KUKA KRL program: Circular.src, Circular.dat

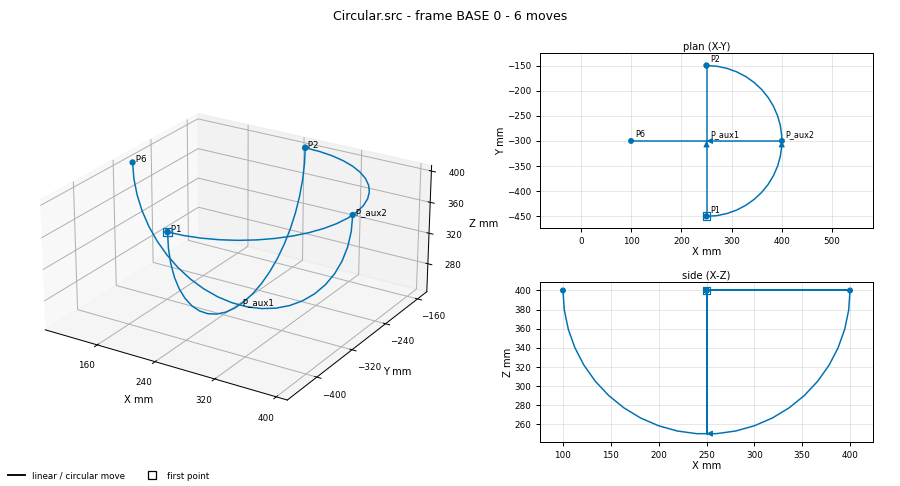
[picture p0: tool path of Circular.src in frame BASE 0, 6 of 10 moves have a stored position in this frame; points joined in program order, loops and branches not executed]
--- Circular.src ---
&ACCESS RVO
&REL 2
&PARAM DISKPATH = KRC:\R1\Program\My_Project
DEF  Circular ( )
;FOLD INI;%{PE}
  ;FOLD BASISTECH INI
    GLOBAL INTERRUPT DECL 3 WHEN $STOPMESS==TRUE DO IR_STOPM ( )
    INTERRUPT ON 3
    BAS (#INITMOV,0 )
  ;ENDFOLD (BASISTECH INI)
  ;FOLD USER INI
    ;Make your modifications here

  ;ENDFOLD (USER INI)
;ENDFOLD (INI)

;FOLD SPTP HOME Vel=100 % DEFAULT ;%{PE}
;FOLD Parameters ;%{h}
;Params IlfProvider=kukaroboter.basistech.inlineforms.movement.spline; Kuka.IsGlobalPoint=False; Kuka.PointName=HOME; Kuka.BlendingEnabled=False; Kuka.MoveDataPtpName=DEFAULT; Kuka.VelocityPtp=100; Kuka.VelocityFieldEnabled=True; Kuka.CurrentCDSetIndex=0; Kuka.MovementParameterFieldEnabled=True; IlfCommand=SPTP
;ENDFOLD
PTP XHOME                                              ;Go to Home position
;ENDFOLD

$BWDSTART = FALSE
PDAT_ACT = PPDATP
FDAT_ACT = FP
BAS(#PTP_PARAMS, 100)
SET_CD_PARAMS(0)


PTP P1                                            ;PTP movement to Point P1
$CIRC_TYPE = #BASE                                ;Set control of circular movement to be BASE related
$ORI_TYPE = #CONSTANT                             ;Set Orientation of the TCP to be CONSTANT
TraceStart("New_KSS_8.5_1.xml", "roll")           ;Start recording trace with the mentioned Trace configuration
CIRC P_aux1, P2, CA 360.0
TraceStop()
PTP XHOME

PTP P3                                            ;PTP movement to Point P3
$CIRC_TYPE = #BASE                                ;Set control of circular movement to be BASE related
$ORI_TYPE = #CONSTANT                             ;Set Orientation of the TCP to be CONSTANT
TraceStart("New_KSS_8.5_1.xml", "yaw")            ;Start recording trace with the mentioned Trace configuration
CIRC P_aux2, P4, CA 360.0
TraceStop()
PTP XHOME

PTP P5                                            ;PTP movement to Point P5
$CIRC_TYPE = #BASE                                ;Set control of circular movement to be BASE related
$ORI_TYPE = #CONSTANT                             ;Set Orientation of the TCP to be CONSTANT
TraceStart("New_KSS_8.5_1.xml", "pitch")          ;Start recording trace with the mentioned Trace configuration
CIRC P_aux3, P6, CA 360.0
TraceStop()

;FOLD SPTP HOME Vel=100 % DEFAULT ;%{PE}
;FOLD Parameters ;%{h}
;Params IlfProvider=kukaroboter.basistech.inlineforms.movement.spline; Kuka.IsGlobalPoint=False; Kuka.PointName=HOME; Kuka.BlendingEnabled=False; Kuka.MoveDataPtpName=DEFAULT; Kuka.VelocityPtp=100; Kuka.VelocityFieldEnabled=True; Kuka.CurrentCDSetIndex=0; Kuka.MovementParameterFieldEnabled=True; IlfCommand=SPTP
;ENDFOLD
PTP XHOME                                              ;Go to Home position
;ENDFOLD

END

--- Circular.dat ---
&ACCESS RVO
&REL 2
&PARAM DISKPATH = KRC:\R1\Program\My_Project
DEFDAT Circular
;FOLD EXTERNAL DECLARATIONS;%{PE}%MKUKATPBASIS,%CEXT,%VCOMMON,%P
;FOLD BASISTECH EXT;%{PE}%MKUKATPBASIS,%CEXT,%VEXT,%P
EXT  BAS (BAS_COMMAND  :IN,REAL  :IN )
DECL INT SUCCESS
;ENDFOLD (BASISTECH EXT)
;FOLD USER EXT;%{E}%MKUKATPUSER,%CEXT,%VEXT,%P
;Make your modifications here

DECL E6AXIS XHOME = {A1 0.0, A2 -110.0, A3 110.0, A4 0.0, A5 0.0, A6 0.0}                  ;Home Position

DECL PDAT PPDATP={VEL 100.000,ACC 100.000,APO_DIST 100.000,APO_MODE #CDIS,GEAR_JERK 100.000,EXAX_IGN 0}     ;Set the kinematic values such as max velocity, max acceleration, etc
DECL FDAT FP={TOOL_NO 14,BASE_NO 0,IPO_FRAME #BASE,POINT2[] " ",TQ_STATE FALSE}                             ;Set the tool and base for coordinate transformation

DECL E6POS P1 = {X 250.0, Y -450.0, Z 400.0, A 0.0, B 45, C 0.0, S 2, T 10}                 ;Point P1
DECL E6POS P_aux1 = {X 250.0, Y -300.0, Z 250.0, A 0.0, B 45, C 0.0, S 2, T 10}             ;Point P_aux1
DECL E6POS P2 = {X 250.0, Y -150.0, Z 400.0, A 0.0, B 45, C 0.0, S 2, T 10}                 ;Point P2

DECL E6POS P3 = {X 250.0, Y -450.0, Z 400.0, A -12.32, B 82.93, C -12.5, S 2, T 10}         ;Point P3
DECL E6POS P_aux2 = {X 400.0, Y -300.0, Z 400.0, A -12.32, B 82.93, C -12.5, S 2, T 10}     ;Point P_aux2
DECL E6POS P4 = {X 250.0, Y -150.0, Z 400.0, A -12.32, B 82.93, C -12.5, S 2, T 10}         ;Point P4

DECL E6POS P5 = {X 400.0, Y -300.0, Z 400.0, A 0.0, B 45.0, C 0.0, S 2, T 10}               ;Point P5
DECL E6POS P_aux3 = {X 250.0, Y -300.0, Z 250.0, A 0.0, B 45.0, C 0.0, S 2, T 10}           ;Point P_aux3
DECL E6POS P6 = {X 100.0, Y -300.0, Z 400.0, A 0.0, B 45.0, C 0.0, S 2, T 10}               ;Point P6


;ENDFOLD (USER EXT)
;ENDFOLD (EXTERNAL DECLARATIONS)
ENDDAT
